// TIA Portal V18 export
DATA_BLOCK "ROBOT_CONV_DB"   // DB3
{ S7_Optimized_Access := 'FALSE' }
   VAR
      input : Array[0..127] of Bool;
      output : Array[0..127] of Bool;
   END_VAR
BEGIN
END_DATA_BLOCK
